# B&R Automation Studio project TrackingSample
Automation Studio 4.10.2.37; technology packages: mappCockpit 5.16.7002, mappMotion 5.16.7500, mappView 5.16.7001

## Configuration Cfg1

CPU 5PC900.TS17-00, AutomationRuntime B4.82, Build 6.3.0, Safety 1.10, Vc V4.33.0

### Task classes (Cpu.sw)
```
Cyclic#1 (cycle 1600 us, tolerance 0 us):
  DeltaCtrl <- Source.Motion.DeltaCtrl.prg
  ConveyorA <- Source.Motion.ConveyorA.prg
  ConveyorB <- Source.Motion.ConveyorB.prg
  ProductDet <- Source.Motion.ProductDetect.prg
  ProductPla <- Source.Motion.ProductPlacement.prg
  Program1 <- (binary)
  ServerP <- (binary)
  ServerR <- (binary)
  UN_Contro2 <- (binary)
DataObjects: McAcpSys, assl1
NcDataObjects: McDriveLog, mainCam, mainCam2, Cam
Binaries: TCData, udbdef, mcacpdrv, McMechSys, McAcpSim, McProfGen, arsvcreg, ArFlatPrv, ArCoal, McPathXT, mvLoader, mCoWebSc, Config_1, ashwd, sysconf, ashwac, asfw, arconfig, Role, iomap, User, Hierarchy, Rob1Ax, CodLim, Rob1AxGr4, CodMec4, Settings, Config, Config_7, Conveyor, CodMec, CodAxGr, Rob1AxGr, Config_5, Config_2, TCLang, Wr_Histor, Al_History, Al_Core, Wr_Core, GroupCore, Ev_Core, TraceConfi, Vis, TriggerCfg, ShuttleCfg, SectorCfg, AssemblyCf, asiol3, Vtrak, TC, User_1, asiol2, FifthAxCfg, PlowHeight, asnxdb3, viApp, Settings_1, viApp2, viApp1, viComp, asiol1, Config_3, asnxdb2, Cod_AxGr, Cod_Lim, Cod_Mec, Rob1_AxGr, Rob1_Ax, asiol4, OpcUaMap, asnxdb1, TriggCfg, Cams, Features, Webx_1, AssemblyCfg, Config_4, UNA, EM00, EM01, EMG, EMA, UN, EM00G, EM00A, EM01G, EM01A, PML
Libraries: DataObj, standard, runtime, astime, MpBase, AsArSdm, asstring, AsBrStr, MTTypes, brsystem, MTFilter, sys_lib, McBase, McAcpTrak, McAxis, McAcpPar, MpAxis, McAcpAx, CamProf, McPureVAx, MTBasics, AsIecCon, powerlnk, AsBrMath, BRIT_Data, MpRobotics, McAxGroup, McPathGen, McProgInt, AsIODiag, McTrkPath, MpPick, McPathSvc, CoTrace, AsZip, FileIO, asarprof, asarlog, AsMem, AsEPL, arssl, AsIO, aruser, ViBase, AsXml, AsTCP, SIKODrvLib, AcpInvLib, AsIOAcc, RVCarousel, AsSafety, MpServer, R_Lib_PM, AsHttp, MpRecipe, R_Lib, AsARCfg, R_Lib_Trak, R_PkML, MpPackML, MpAlarmX, ArUnitText, R_Siko, R_Carousel, areventlog
```

### Hardware
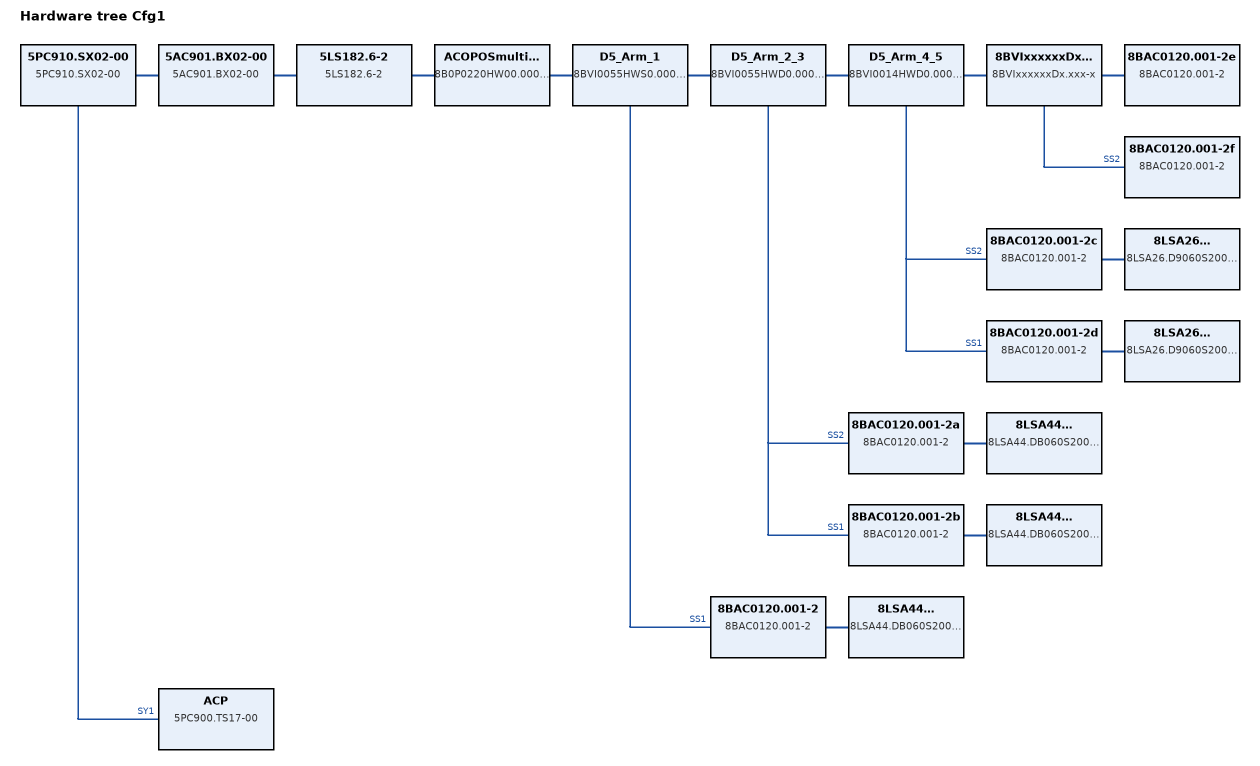
```
5AC901.BX02-00 : 5AC901.BX02-00 v1.0.1.0  [SY -> 5PC910.SX02-00.SY3]
5LS182.6-2 : 5LS182.6-2 v1.7.0.0  [SL -> 5AC901.BX02-00.SL1]
  Connector IF1:
    MtuSize = 1500
    DNAConfiguration = manual
    CycleTime = 1600
    EplNatSubnet = 192.168.102.0
    Channel1
    ChannelID1 = McAcpBroadcast
    ChannelType1 = OCTET[40]
    InternetAddress = 192.168.200.240
    SubnetMask = 255.255.255.0
5PC910.SX02-00 : 5PC910.SX02-00 v2.0.3.0
  Connector IF1:
    AssignedOperatingSystem = ARemb
  Connector IF3:
    AssignedOperatingSystem = ARemb
    ActivateDevice = 1
    Mode = Manual
    InternetAddress = 192.168.150.227
    SubnetMask = 255.255.255.0
  Connector IF4:
    AssignedOperatingSystem = ARemb
    ActivateDevice = 1
    Mode = Manual
    InternetAddress = 192.168.13.2
    SubnetMask = 255.255.255.0
  Connector IF5:
    AssignedOperatingSystem = ARemb
  Connector IF6:
    AssignedOperatingSystem = ARemb
  Connector IF7:
    AssignedOperatingSystem = ARemb
  Connector IF8:
    AssignedOperatingSystem = ARemb
  Connector IF9:
    AssignedOperatingSystem = ARemb
8BAC0120.001-2 : 8BAC0120.001-2 v2.2.0.0  [SS -> D5_Arm_1.SS1]
  PlugInType = Encoder
  McAcoposTypeID = AcoposMultiPlugInConfig
8BAC0120.001-2a : 8BAC0120.001-2 v2.2.0.0  [SS -> D5_Arm_2_3.SS2]
  PlugInType = Encoder
  McAcoposTypeID = AcoposMultiPlugInConfig
8BAC0120.001-2b : 8BAC0120.001-2 v2.2.0.0  [SS -> D5_Arm_2_3.SS1]
  PlugInType = Encoder
  McAcoposTypeID = AcoposMultiPlugInConfig
8BAC0120.001-2c : 8BAC0120.001-2 v2.2.0.0  [SS -> D5_Arm_4_5.SS2]
  PlugInType = Encoder
  McAcoposTypeID = AcoposMultiPlugInConfig
8BAC0120.001-2d : 8BAC0120.001-2 v2.2.0.0  [SS -> D5_Arm_4_5.SS1]
  PlugInType = Encoder
  McAcoposTypeID = AcoposMultiPlugInConfig
8BAC0120.001-2e : 8BAC0120.001-2 v2.2.0.0  [SS -> 8BVIxxxxxxDx.xxx-x2.SS1]
  PlugInType = Encoder
  McAcoposTypeID = AcoposMultiPlugInConfig
8BAC0120.001-2f : 8BAC0120.001-2 v2.2.0.0  [SS -> 8BVIxxxxxxDx.xxx-x2.SS2]
  PlugInType = Encoder
  McAcoposTypeID = AcoposMultiPlugInConfig
8BVIxxxxxxDx.xxx-x2 : 8BVIxxxxxxDx.xxx-x v2.3.0.0  [PLK1 -> D5_Arm_4_5.PLK2 (NodeNumber=7) [Cable Type=PowerlinkCable, Length=10, Version=1.0.0.3]]
  OrderNumber = 8BVI0014HWD0.000-1
  DriveConfiguration/Module:
    McAcoposTypeID = AcoposMultiDConfig
    ActivateACOPOSSimulationOnPLC = 0
    PowerSupply = DCBusVoltage
  DriveConfiguration/Module/PowerSupply:
    BusVoltage = 550
  DriveConfiguration/Channel[1]/RealAxis:
    AxisReference = gAxisConvB
  DriveConfiguration/Channel[1]/RealAxis/MechanicalElements/Gearbox:
    InputIsReadOnly = 0
    Input = 1
    OutputIsReadOnly = 0
    Output = 10
  DriveConfiguration/Channel[1]/RealAxis/MechanicalElements/RotaryToLinearTransformation:
    ReferenceDistanceIsReadOnly = 0
    ReferenceDistance = 3
  DriveConfiguration/Channel[1]/RealAxis/Controller:
    ModeIsReadOnly = 0
    Mode = PositionController
  DriveConfiguration/Channel[1]/RealAxis/Controller/Mode/Position:
    ProportionalGain = 460
    IntegrationTime = 0.0
    PredictionTime = 0.0004
    TotalDelayTime = 0.0004
  DriveConfiguration/Channel[1]/RealAxis/Controller/Mode/Speed:
    ProportionalGainIsReadOnly = 0
    ProportionalGain = 0.6
    IntegrationTimeIsReadOnly = 0
    IntegrationTime = 0.0
    FilterTimeIsReadOnly = 0
    FilterTime = 0.0
  DriveConfiguration/Channel[1]/RealAxis/Controller/Mode/LoopFilters:
    LoopFilter1 = NotUsed
    LoopFilter2 = NotUsed
    LoopFilter3 = NotUsed
  DriveConfiguration/Channel[1]/RealAxis/Homing:
    Mode = Direct
  DriveConfiguration/Channel[1]/RealAxis/Homing/Mode:
    Position = 0.0
    ReferencePulse = NotUsed
  DriveConfiguration/Channel[1]/RealAxis/Homing:
    RestorePositionVariable = 
  DriveConfiguration/Channel[1]/RealAxis/StopReaction:
    Quickstop = DecelerationLimit
    DriveError = DecelerationLimit
  DriveConfiguration/Channel[1]/RealAxis/MovementErrorLimits:
    PositionError = 1.0
    VelocityErrorMonitoring = Automatic1
  DriveConfiguration/Channel[1]/RealAxis:
    JerkFilter = NotUsed
  DriveConfiguration/Channel[1]/RealAxis/DigitalInputs/HomingSwitch:
    Source = NotUsed
    Level = High
  DriveConfiguration/Channel[1]/RealAxis/DigitalInputs/PositiveLimitSwitch:
    Source = NotUsed
    Level = High
  DriveConfiguration/Channel[1]/RealAxis/DigitalInputs/NegativeLimitSwitch:
    Source = NotUsed
    Level = High
  DriveConfiguration/Channel[1]/RealAxis/DigitalInputs/Trigger1:
    Source = X2Trigger1
    Level = High
  DriveConfiguration/Channel[1]/RealAxis/DigitalInputs/Trigger2:
    Source = X2Trigger2
    Level = High
  DriveConfiguration/Channel[1]/RealAxis/DigitalInputs/Quickstop:
    Input = Trigger2
  DriveConfiguration/Channel[1]/RealAxis/Simulation:
    SimulationModeOnPLC = SetValueGeneration
    SimulationModeOnACOPOS = NotUsed
  DriveConfiguration/Channel[1]:
    ExternalEncoderAxis = NotUsed
  DriveConfiguration/Channel[2]/RealAxis:
    AxisReference = gAxisConvA
  DriveConfiguration/Channel[2]/RealAxis/MechanicalElements/Gearbox:
    InputIsReadOnly = 0
    Input = 1
    OutputIsReadOnly = 0
    Output = 10
  DriveConfiguration/Channel[2]/RealAxis/MechanicalElements/RotaryToLinearTransformation:
    ReferenceDistanceIsReadOnly = 0
    ReferenceDistance = 3
  DriveConfiguration/Channel[2]/RealAxis/Controller:
    ModeIsReadOnly = 0
    Mode = PositionController
  DriveConfiguration/Channel[2]/RealAxis/Controller/Mode/Position:
    ProportionalGain = 435
    IntegrationTime = 0.0
    PredictionTime = 0.0004
    TotalDelayTime = 0.0004
  DriveConfiguration/Channel[2]/RealAxis/Controller/Mode/Speed:
    ProportionalGainIsReadOnly = 0
    ProportionalGain = 0.55
    IntegrationTimeIsReadOnly = 0
    IntegrationTime = 0.0
    FilterTimeIsReadOnly = 0
    FilterTime = 0.0
  DriveConfiguration/Channel[2]/RealAxis/Controller/Mode/LoopFilters:
    LoopFilter1 = NotUsed
    LoopFilter2 = NotUsed
    LoopFilter3 = NotUsed
  DriveConfiguration/Channel[2]/RealAxis/Homing:
    Mode = Direct
  DriveConfiguration/Channel[2]/RealAxis/Homing/Mode:
    Position = 0.0
    ReferencePulse = NotUsed
  DriveConfiguration/Channel[2]/RealAxis/Homing:
    RestorePositionVariable = 
  DriveConfiguration/Channel[2]/RealAxis/StopReaction:
    Quickstop = DecelerationLimit
    DriveError = DecelerationLimit
  DriveConfiguration/Channel[2]/RealAxis/MovementErrorLimits:
    PositionError = 1.0
    VelocityErrorMonitoring = Automatic1
  DriveConfiguration/Channel[2]/RealAxis:
    JerkFilter = NotUsed
  DriveConfiguration/Channel[2]/RealAxis/DigitalInputs/HomingSwitch:
    Source = NotUsed
    Level = High
  DriveConfiguration/Channel[2]/RealAxis/DigitalInputs/PositiveLimitSwitch:
    Source = NotUsed
    Level = High
  DriveConfiguration/Channel[2]/RealAxis/DigitalInputs/NegativeLimitSwitch:
    Source = NotUsed
    Level = High
  DriveConfiguration/Channel[2]/RealAxis/DigitalInputs/Trigger1:
    Source = X2Trigger1
    Level = High
  DriveConfiguration/Channel[2]/RealAxis/DigitalInputs/Trigger2:
    Source = X2Trigger2
    Level = High
  DriveConfiguration/Channel[2]/RealAxis/DigitalInputs/Quickstop:
    Input = Trigger2
  DriveConfiguration/Channel[2]/RealAxis/Simulation:
    SimulationModeOnPLC = SetValueGeneration
    SimulationModeOnACOPOS = NotUsed
  DriveConfiguration/Channel[2]:
    ExternalEncoderAxis = NotUsed
8LSA26.D9060S200-3 : 8LSA26.D9060S200-3 v1.0.7.40  [EC -> 8BAC0120.001-2d.EC; MT -> D5_Arm_4_5.MT1]
8LSA26.D9060S200-3a : 8LSA26.D9060S200-3 v1.0.7.40  [EC -> 8BAC0120.001-2c.EC; MT -> D5_Arm_4_5.MT2]
8LSA44.DB060S200-3 : 8LSA44.DB060S200-3 v1.0.9.37  [EC -> 8BAC0120.001-2.EC; MT -> D5_Arm_1.MT1]
8LSA44.DB060S200-3a : 8LSA44.DB060S200-3 v1.0.9.37  [EC -> 8BAC0120.001-2a.EC; MT -> D5_Arm_2_3.MT2]
8LSA44.DB060S200-3b : 8LSA44.DB060S200-3 v1.0.9.37  [EC -> 8BAC0120.001-2b.EC; MT -> D5_Arm_2_3.MT1]
ACOPOSmulti_Rack_PS : 8B0P0220HW00.000-1 v2.3.0.0  [PLK1 -> 5LS182.6-2.IF1 (NodeNumber=100) [Cable Type=PowerlinkCable, Length=10, Version=1.0.0.3]; PLK2 -> D5_Arm_1.PLK1 (NodeNumber=100) [Cable Type=PowerlinkCable, Length=10, Version=1.0.0.3]]
  DriveConfiguration/Module:
    McAcoposTypeID = AcoposMultiPSMpConfig
    ActivateACOPOSSimulationOnPLC = 0
  DriveConfiguration/Channel[1]/PowerSection:
    AxisReference = gRobPS
  DriveConfiguration/Channel[1]/ChannelFeatures:
    FeatureRef[1] = Feature_AcpParTable
ACP : 5PC900.TS17-00 v2.1.0.0  [SY -> 5PC910.SX02-00.SY1]
  ConfigurationID = Betel
  UserPartitionSize = 10
  Simulation = 1
  RemMemDevice = PCI.1.LS182.SRAM
  RemMemSize = 10000
  PermanentPvSize = 9000
  RemanentGlobalPvSize = 100
  VolatileGlobalPvSize = 4000000
  ClearNVMemoryAfterCFChange = 1
  TimerDeviceType = EPLX2X
  TimerDevice = 5LS182.6-2.IF1
  IdleTaskClass = 4
  TaskClassIdleTime = 3200
  Cyclic1Duration = 1600
  Cyclic1Tolerance = 0
  Cyclic1Stack = 1000000
  Cyclic1Output = 1
  Cyclic2Duration = 19200
  Cyclic2Tolerance = 19200
  Cyclic3Duration = 48000
  Cyclic3Tolerance = 48000
  Cyclic4Duration = 99200
  Cyclic4Tolerance = 99200
  Cyclic6Duration = 499200
  Cyclic6Tolerance = 499200
  Cyclic8Duration = 16000
  FileDevice1
  FileDeviceName1 = CNC_Programs
  FileDevicePath1 = C:\projects\MCR\TrackingSample\Logical\Source\Motion\RobotProgram
  TimeZone = 140
  ActivateDaylightSavingTime = 1
  FtpUser1
  FtpUsername1 = ronchi
  FtpUserPassword1 = Qr4mnGyRDGFj5/UnqR7ZzE2TygV13U3viQDWrGQj2Tc=
  FtpUserSalt1 = 2ZufkTNm
  FTPAccessRight1 = 0
  ActivateOpcUa = 1
  OpcUa_AuthenticationSecurityPolicy_EnableNone = 1
  OpcUa_AuthenticationSecurityPolicy_EnableBasic128Rsa15 = 1
  OpcUa_Security_AdminRole = Everyone
  OpcUa_Limits_MonitoredItemsPerSubscription = 5000
  OpcUaMaxSubsEventQueueSize = 5000
  OpcUaInformationModels_PV_Version = 1
D5_Arm_1 : 8BVI0055HWS0.000-1 v2.2.0.0  [PLK1 -> ACOPOSmulti_Rack_PS.PLK2 [Cable Type=PowerlinkCable, Length=10, Version=1.0.0.3]; PLK2 -> D5_Arm_2_3.PLK1 [Cable Type=PowerlinkCable, Length=10, Version=1.0.0.3]]
  DriveConfiguration/Module:
    McAcoposTypeID = AcoposMultiDConfig
    ActivateACOPOSSimulationOnPLC = 0
  DriveConfiguration/Module/PowerSupply:
    PowerSupplyModuleReference = gRobPS
  DriveConfiguration/Channel[1]/RealAxis:
    AxisReference = gR1_AxisQ1
  DriveConfiguration/Channel[1]/RealAxis/MechanicalElements/Gearbox:
    InputIsReadOnly = 0
    Input = 31
    OutputIsReadOnly = 0
    Output = 1
  DriveConfiguration/Channel[1]/RealAxis/MechanicalElements/RotaryToLinearTransformation:
    ReferenceDistanceIsReadOnly = 0
    ReferenceDistance = 1
  DriveConfiguration/Channel[1]/RealAxis/Controller:
    ModeIsReadOnly = 0
    Mode = PositionController
  DriveConfiguration/Channel[1]/RealAxis/Controller/Mode/Position:
    ProportionalGain = 150
    IntegrationTime = 0.0
    PredictionTime = 0.0004
    TotalDelayTime = 0.0004
  DriveConfiguration/Channel[1]/RealAxis/Controller/Mode/Speed:
    ProportionalGainIsReadOnly = 0
    ProportionalGain = 5
    IntegrationTimeIsReadOnly = 0
    IntegrationTime = 0.0
    FilterTimeIsReadOnly = 0
    FilterTime = 0.0
  DriveConfiguration/Channel[1]/RealAxis/Controller/Mode/LoopFilters:
    LoopFilter1 = NotUsed
    LoopFilter2 = NotUsed
    LoopFilter3 = NotUsed
  DriveConfiguration/Channel[1]/RealAxis/Homing:
    Mode = RestorePosition
    RestorePositionVariable = ::HomePos_R1[0]
  DriveConfiguration/Channel[1]/RealAxis/StopReaction:
    Quickstop = DecelerationLimit
    DriveError = DecelerationLimit
  DriveConfiguration/Channel[1]/RealAxis/MovementErrorLimits:
    PositionError = 1.0
    VelocityErrorMonitoring = Automatic1
  DriveConfiguration/Channel[1]/RealAxis:
    JerkFilter = Used
  DriveConfiguration/Channel[1]/RealAxis/JerkFilter:
    JerkTime = 0.02
  DriveConfiguration/Channel[1]/RealAxis/DigitalInputs/HomingSwitch:
    Source = NotUsed
    Level = High
  DriveConfiguration/Channel[1]/RealAxis/DigitalInputs/PositiveLimitSwitch:
    Source = NotUsed
    Level = High
  DriveConfiguration/Channel[1]/RealAxis/DigitalInputs/NegativeLimitSwitch:
    Source = NotUsed
    Level = High
  DriveConfiguration/Channel[1]/RealAxis/DigitalInputs/Trigger1:
    Level = High
  DriveConfiguration/Channel[1]/RealAxis/DigitalInputs/Trigger2:
    Level = High
  DriveConfiguration/Channel[1]/RealAxis/DigitalInputs/Quickstop:
    Input = Trigger2
  DriveConfiguration/Channel[1]/RealAxis/Simulation:
    SimulationModeOnPLC = SetValueGeneration
    SimulationModeOnACOPOS = NotUsed
  DriveConfiguration/Channel[2]/RealAxis:
    AxisReference = 
  DriveConfiguration/Channel[2]/RealAxis/MechanicalElements/Gearbox:
    InputIsReadOnly = 0
    Input = 1
    OutputIsReadOnly = 0
    Output = 1
  DriveConfiguration/Channel[2]/RealAxis/MechanicalElements/RotaryToLinearTransformation:
    ReferenceDistanceIsReadOnly = 0
    ReferenceDistance = 1
  DriveConfiguration/Channel[2]/RealAxis/Controller:
    ModeIsReadOnly = 0
    Mode = PositionController
  DriveConfiguration/Channel[2]/RealAxis/Controller/Mode/Position:
    ProportionalGain = 50.0
    IntegrationTime = 0.0
    PredictionTime = 0.0004
    TotalDelayTime = 0.0004
  DriveConfiguration/Channel[2]/RealAxis/Controller/Mode/Speed:
    ProportionalGainIsReadOnly = 0
    ProportionalGain = 2.0
    IntegrationTimeIsReadOnly = 0
    IntegrationTime = 0.0
    FilterTimeIsReadOnly = 0
    FilterTime = 0.0
  DriveConfiguration/Channel[2]/RealAxis/Controller/Mode/LoopFilters:
    LoopFilter1 = NotUsed
    LoopFilter2 = NotUsed
    LoopFilter3 = NotUsed
  DriveConfiguration/Channel[2]/RealAxis/Homing:
    Mode = Direct
  DriveConfiguration/Channel[2]/RealAxis/Homing/Mode:
    Position = 0.0
    ReferencePulse = NotUsed
  DriveConfiguration/Channel[2]/RealAxis/Homing:
    RestorePositionVariable = 
  DriveConfiguration/Channel[2]/RealAxis/StopReaction:
    Quickstop = DecelerationLimit
    DriveError = DecelerationLimit
  DriveConfiguration/Channel[2]/RealAxis/MovementErrorLimits:
    PositionError = 1.0
    VelocityErrorMonitoring = Automatic1
  DriveConfiguration/Channel[2]/RealAxis:
    JerkFilter = NotUsed
  DriveConfiguration/Channel[2]/RealAxis/DigitalInputs/HomingSwitch:
    Source = NotUsed
    Level = High
  DriveConfiguration/Channel[2]/RealAxis/DigitalInputs/PositiveLimitSwitch:
    Source = NotUsed
    Level = High
  DriveConfiguration/Channel[2]/RealAxis/DigitalInputs/NegativeLimitSwitch:
    Source = NotUsed
    Level = High
  DriveConfiguration/Channel[2]/RealAxis/DigitalInputs/Trigger1:
    Level = High
  DriveConfiguration/Channel[2]/RealAxis/DigitalInputs/Trigger2:
    Level = High
  DriveConfiguration/Channel[2]/RealAxis/DigitalInputs/Quickstop:
    Input = Trigger2
  DriveConfiguration/Channel[2]/RealAxis/Simulation:
    SimulationModeOnPLC = SetValueGeneration
    SimulationModeOnACOPOS = NotUsed
D5_Arm_2_3 : 8BVI0055HWD0.000-1 v2.2.0.0  [PLK1 -> D5_Arm_1.PLK2 [Cable Type=PowerlinkCable, Length=10, Version=1.0.0.3]; PLK2 -> D5_Arm_4_5.PLK1 [Cable Type=PowerlinkCable, Length=10, Version=1.0.0.3]; MT2 -> 8LSA44.DB060S200-3a.MT]
  DriveConfiguration/Module:
    McAcoposTypeID = AcoposMultiDConfig
    ActivateACOPOSSimulationOnPLC = 0
  DriveConfiguration/Module/PowerSupply:
    PowerSupplyModuleReference = gRobPS
  DriveConfiguration/Channel[1]/RealAxis:
    AxisReference = gR1_AxisQ3
  DriveConfiguration/Channel[1]/RealAxis/MechanicalElements/Gearbox:
    InputIsReadOnly = 0
    Input = 31
    OutputIsReadOnly = 0
    Output = 1
  DriveConfiguration/Channel[1]/RealAxis/MechanicalElements/RotaryToLinearTransformation:
    ReferenceDistanceIsReadOnly = 0
    ReferenceDistance = 1
  DriveConfiguration/Channel[1]/RealAxis/Controller:
    ModeIsReadOnly = 0
    Mode = PositionController
  DriveConfiguration/Channel[1]/RealAxis/Controller/Mode/Position:
    ProportionalGain = 150
    IntegrationTime = 0.0
    PredictionTime = 0.0004
    TotalDelayTime = 0.0004
  DriveConfiguration/Channel[1]/RealAxis/Controller/Mode/Speed:
    ProportionalGainIsReadOnly = 0
    ProportionalGain = 5
    IntegrationTimeIsReadOnly = 0
    IntegrationTime = 0.0
    FilterTimeIsReadOnly = 0
    FilterTime = 0.0
  DriveConfiguration/Channel[1]/RealAxis/Controller/Mode/LoopFilters:
    LoopFilter1 = NotUsed
    LoopFilter2 = NotUsed
    LoopFilter3 = NotUsed
  DriveConfiguration/Channel[1]/RealAxis/Homing:
    Mode = RestorePosition
    RestorePositionVariable = ::HomePos_R1[2]
  DriveConfiguration/Channel[1]/RealAxis/StopReaction:
    Quickstop = DecelerationLimit
    DriveError = DecelerationLimit
  DriveConfiguration/Channel[1]/RealAxis/MovementErrorLimits:
    PositionError = 1.0
    VelocityErrorMonitoring = Automatic1
  DriveConfiguration/Channel[1]/RealAxis:
    JerkFilter = Used
  DriveConfiguration/Channel[1]/RealAxis/JerkFilter:
    JerkTime = 0.02
  DriveConfiguration/Channel[1]/RealAxis/DigitalInputs/HomingSwitch:
    Source = NotUsed
    Level = High
  DriveConfiguration/Channel[1]/RealAxis/DigitalInputs/PositiveLimitSwitch:
    Source = NotUsed
    Level = High
  DriveConfiguration/Channel[1]/RealAxis/DigitalInputs/NegativeLimitSwitch:
    Source = NotUsed
    Level = High
  DriveConfiguration/Channel[1]/RealAxis/DigitalInputs/Trigger1:
    Level = High
  DriveConfiguration/Channel[1]/RealAxis/DigitalInputs/Trigger2:
    Level = High
  DriveConfiguration/Channel[1]/RealAxis/DigitalInputs/Quickstop:
    Input = Trigger2
  DriveConfiguration/Channel[1]/RealAxis/Simulation:
    SimulationModeOnPLC = SetValueGeneration
    SimulationModeOnACOPOS = NotUsed
  DriveConfiguration/Channel[2]/RealAxis:
    AxisReference = gR1_AxisQ2
  DriveConfiguration/Channel[2]/RealAxis/MechanicalElements/Gearbox:
    InputIsReadOnly = 0
    Input = 31
    OutputIsReadOnly = 0
    Output = 1
  DriveConfiguration/Channel[2]/RealAxis/MechanicalElements/RotaryToLinearTransformation:
    ReferenceDistanceIsReadOnly = 0
    ReferenceDistance = 1
  DriveConfiguration/Channel[2]/RealAxis/Controller:
    ModeIsReadOnly = 0
    Mode = PositionController
  DriveConfiguration/Channel[2]/RealAxis/Controller/Mode/Position:
    ProportionalGain = 150
    IntegrationTime = 0.0
    PredictionTime = 0.0004
    TotalDelayTime = 0.0004
  DriveConfiguration/Channel[2]/RealAxis/Controller/Mode/Speed:
    ProportionalGainIsReadOnly = 0
    ProportionalGain = 5
    IntegrationTimeIsReadOnly = 0
    IntegrationTime = 0.0
    FilterTimeIsReadOnly = 0
    FilterTime = 0.0
  DriveConfiguration/Channel[2]/RealAxis/Controller/Mode/LoopFilters:
    LoopFilter1 = NotUsed
    LoopFilter2 = NotUsed
    LoopFilter3 = NotUsed
  DriveConfiguration/Channel[2]/RealAxis/Homing:
    Mode = RestorePosition
    RestorePositionVariable = ::HomePos_R1[1]
  DriveConfiguration/Channel[2]/RealAxis/StopReaction:
    Quickstop = DecelerationLimit
    DriveError = DecelerationLimit
  DriveConfiguration/Channel[2]/RealAxis/MovementErrorLimits:
    PositionError = 1.0
    VelocityErrorMonitoring = Automatic1
  DriveConfiguration/Channel[2]/RealAxis:
    JerkFilter = Used
  DriveConfiguration/Channel[2]/RealAxis/JerkFilter:
    JerkTime = 0.02
  DriveConfiguration/Channel[2]/RealAxis/DigitalInputs/HomingSwitch:
    Source = NotUsed
    Level = High
  DriveConfiguration/Channel[2]/RealAxis/DigitalInputs/PositiveLimitSwitch:
    Source = NotUsed
    Level = High
  DriveConfiguration/Channel[2]/RealAxis/DigitalInputs/NegativeLimitSwitch:
    Source = NotUsed
    Level = High
  DriveConfiguration/Channel[2]/RealAxis/DigitalInputs/Trigger1:
    Level = High
  DriveConfiguration/Channel[2]/RealAxis/DigitalInputs/Trigger2:
    Level = High
  DriveConfiguration/Channel[2]/RealAxis/DigitalInputs/Quickstop:
    Input = Trigger2
  DriveConfiguration/Channel[2]/RealAxis/Simulation:
    SimulationModeOnPLC = SetValueGeneration
    SimulationModeOnACOPOS = NotUsed
D5_Arm_4_5 : 8BVI0014HWD0.000-1 v2.2.0.0  [PLK1 -> D5_Arm_2_3.PLK2 [Cable Type=PowerlinkCable, Length=10, Version=1.0.0.3]; PLK2 -> 8BVIxxxxxxDx.xxx-x2.PLK1 [Cable Type=PowerlinkCable, Length=10, Version=1.0.0.3]; MT2 -> 8LSA26.D9060S200-3a.MT]
  DriveConfiguration/Module:
    McAcoposTypeID = AcoposMultiDConfig
    ActivateACOPOSSimulationOnPLC = 0
  DriveConfiguration/Module/PowerSupply:
    PowerSupplyModuleReference = gRobPS
  DriveConfiguration/Channel[1]/RealAxis:
    AxisReference = gR1_AxisQC
  DriveConfiguration/Channel[1]/RealAxis/MechanicalElements/Gearbox:
    InputIsReadOnly = 0
    Input = 20
    OutputIsReadOnly = 0
    Output = 1
  DriveConfiguration/Channel[1]/RealAxis/MechanicalElements/RotaryToLinearTransformation:
    ReferenceDistanceIsReadOnly = 0
    ReferenceDistance = 1
  DriveConfiguration/Channel[1]/RealAxis/Controller:
    ModeIsReadOnly = 0
    Mode = PositionController
  DriveConfiguration/Channel[1]/RealAxis/Controller/Mode/Position:
    ProportionalGain = 150
    IntegrationTime = 0.0
    PredictionTime = 0.0004
    TotalDelayTime = 0.0004
  DriveConfiguration/Channel[1]/RealAxis/Controller/Mode/Speed:
    ProportionalGainIsReadOnly = 0
    ProportionalGain = 0.6
    IntegrationTimeIsReadOnly = 0
    IntegrationTime = 0.0
    FilterTimeIsReadOnly = 0
    FilterTime = 0.0
  DriveConfiguration/Channel[1]/RealAxis/Controller/Mode/LoopFilters:
    LoopFilter1 = NotUsed
    LoopFilter2 = NotUsed
    LoopFilter3 = NotUsed
  DriveConfiguration/Channel[1]/RealAxis/Homing:
    Mode = RestorePosition
    RestorePositionVariable = ::HomePos_R1[3]
  DriveConfiguration/Channel[1]/RealAxis/StopReaction:
    Quickstop = DecelerationLimit
    DriveError = DecelerationLimit
  DriveConfiguration/Channel[1]/RealAxis/MovementErrorLimits:
    PositionError = 1.0
    VelocityErrorMonitoring = Automatic1
  DriveConfiguration/Channel[1]/RealAxis:
    JerkFilter = Used
  DriveConfiguration/Channel[1]/RealAxis/JerkFilter:
    JerkTime = 0.01
  DriveConfiguration/Channel[1]/RealAxis/DigitalInputs/HomingSwitch:
    Source = NotUsed
    Level = High
  DriveConfiguration/Channel[1]/RealAxis/DigitalInputs/PositiveLimitSwitch:
    Source = NotUsed
    Level = High
  DriveConfiguration/Channel[1]/RealAxis/DigitalInputs/NegativeLimitSwitch:
    Source = NotUsed
    Level = High
  DriveConfiguration/Channel[1]/RealAxis/DigitalInputs/Trigger1:
    Level = High
  DriveConfiguration/Channel[1]/RealAxis/DigitalInputs/Trigger2:
    Level = High
  DriveConfiguration/Channel[1]/RealAxis/DigitalInputs/Quickstop:
    Input = Trigger2
  DriveConfiguration/Channel[1]/RealAxis/Simulation:
    SimulationModeOnPLC = SetValueGeneration
    SimulationModeOnACOPOS = NotUsed
  DriveConfiguration/Channel[2]/RealAxis:
    AxisReference = gR1_AxisQA
  DriveConfiguration/Channel[2]/RealAxis/MechanicalElements/Gearbox:
    InputIsReadOnly = 0
    Input = 20
    OutputIsReadOnly = 0
    Output = 1
  DriveConfiguration/Channel[2]/RealAxis/MechanicalElements/RotaryToLinearTransformation:
    ReferenceDistanceIsReadOnly = 0
    ReferenceDistance = 1
  DriveConfiguration/Channel[2]/RealAxis/Controller:
    ModeIsReadOnly = 0
    Mode = PositionController
  DriveConfiguration/Channel[2]/RealAxis/Controller/Mode/Position:
    ProportionalGain = 150
    IntegrationTime = 0.0
    PredictionTime = 0.0004
    TotalDelayTime = 0.0004
  DriveConfiguration/Channel[2]/RealAxis/Controller/Mode/Speed:
    ProportionalGainIsReadOnly = 0
    ProportionalGain = 0.6
    IntegrationTimeIsReadOnly = 0
    IntegrationTime = 0.0
    FilterTimeIsReadOnly = 0
    FilterTime = 0.0
  DriveConfiguration/Channel[2]/RealAxis/Controller/Mode/LoopFilters:
    LoopFilter1 = NotUsed
    LoopFilter2 = NotUsed
    LoopFilter3 = NotUsed
  DriveConfiguration/Channel[2]/RealAxis/Homing:
    Mode = RestorePosition
    RestorePositionVariable = ::HomePos_R1[4]
  DriveConfiguration/Channel[2]/RealAxis/StopReaction:
    Quickstop = DecelerationLimit
    DriveError = DecelerationLimit
  DriveConfiguration/Channel[2]/RealAxis/MovementErrorLimits:
    PositionError = 1.0
    VelocityErrorMonitoring = Automatic1
  DriveConfiguration/Channel[2]/RealAxis:
    JerkFilter = Used
  DriveConfiguration/Channel[2]/RealAxis/JerkFilter:
    JerkTime = 0.01
  DriveConfiguration/Channel[2]/RealAxis/DigitalInputs/HomingSwitch:
    Source = NotUsed
    Level = High
  DriveConfiguration/Channel[2]/RealAxis/DigitalInputs/PositiveLimitSwitch:
    Source = NotUsed
    Level = High
  DriveConfiguration/Channel[2]/RealAxis/DigitalInputs/NegativeLimitSwitch:
    Source = NotUsed
    Level = High
  DriveConfiguration/Channel[2]/RealAxis/DigitalInputs/Trigger1:
    Level = High
  DriveConfiguration/Channel[2]/RealAxis/DigitalInputs/Trigger2:
    Level = High
  DriveConfiguration/Channel[2]/RealAxis/DigitalInputs/Quickstop:
    Input = Trigger2
  DriveConfiguration/Channel[2]/RealAxis/Simulation:
    SimulationModeOnPLC = SetValueGeneration
    SimulationModeOnACOPOS = NotUsed
```

### Config.mappmotioncfg - ACP/mappMotion/Config.mappmotioncfg
```
Element MappMotionConfiguration (Type=mappmotioncfg)
  Processing:
    ProcessingTaskClass = 1
  Logger:
    SelectiveLogging = Used
      AdministrativeCommands = Suppressed
      MovementCommands = Visible
      InformationalCommands = Suppressed
      SuppressSubcomponents = Inactive
```

### Config_5.axis - ACP/mappMotion/Config_5.axis
```
Element gAxisConvA (Type=axis)
  BaseTypeIsReadOnly = 0
  BaseType = LinearPeriodic
    MeasurementUnit = 5066068
    MeasurementResolutionIsReadOnly = 0
    MeasurementResolution = 0.001
    CountDirectionIsReadOnly = 0
    CountDirection = Standard
    PeriodSettings:
      Period = 1200
  MovementLimitsIsReadOnly = 0
  MovementLimits = Internal
    Position:
      LowerLimitMin = -1.79769313486231E308
      UpperLimitMax = 1.79769313486231E308
      LowerLimit = -1000.0
      UpperLimit = 1000.0
    VelocityIsReadOnly = 0
    Velocity:
      VelocityMax = 3.4E38
      Velocity = 2000
    AccelerationIsReadOnly = 0
    Acceleration:
      AccelerationMax = 3.4E38
      Acceleration = 5000
    DecelerationIsReadOnly = 0
    Deceleration:
      DecelerationMax = 3.4E38
      Deceleration = 5000
  Alarms = None
```

### Conveyor.axis - ACP/mappMotion/Conveyor.axis
```
Element gAxisConvB (Type=axis)
  BaseTypeIsReadOnly = 0
  BaseType = LinearPeriodic
    MeasurementUnit = 5066068
    MeasurementResolutionIsReadOnly = 0
    MeasurementResolution = 0.001
    CountDirectionIsReadOnly = 0
    CountDirection = Standard
    PeriodSettings:
      Period = 1200
  MovementLimitsIsReadOnly = 0
  MovementLimits = Internal
    Position:
      LowerLimitMin = -1.79769313486231E308
      UpperLimitMax = 1.79769313486231E308
      LowerLimit = -1000.0
      UpperLimit = 1000.0
    VelocityIsReadOnly = 0
    Velocity:
      VelocityMax = 3.4E38
      Velocity = 2000
    AccelerationIsReadOnly = 0
    Acceleration:
      AccelerationMax = 3.4E38
      Acceleration = 5000
    DecelerationIsReadOnly = 0
    Deceleration:
      DecelerationMax = 3.4E38
      Deceleration = 5000
  Alarms = None
Element gAxisConvA (Type=axis)
  BaseTypeIsReadOnly = 0
  BaseType = LinearPeriodic
    MeasurementUnit = 5066068
    MeasurementResolutionIsReadOnly = 0
    MeasurementResolution = 0.001
    CountDirectionIsReadOnly = 0
    CountDirection = Standard
    PeriodSettings:
      Period = 1200
  MovementLimitsIsReadOnly = 0
  MovementLimits = Internal
    Position:
      LowerLimitMin = -1.79769313486231E308
      UpperLimitMax = 1.79769313486231E308
      LowerLimit = -1000.0
      UpperLimit = 1000.0
    VelocityIsReadOnly = 0
    Velocity:
      VelocityMax = 3.4E38
      Velocity = 2000
    AccelerationIsReadOnly = 0
    Acceleration:
      AccelerationMax = 3.4E38
      Acceleration = 5000
    DecelerationIsReadOnly = 0
    Deceleration:
      DecelerationMax = 3.4E38
      Deceleration = 5000
  Alarms = None
```

### CodLim.limitset - ACP/mappMotion/Rob/Codian_4ax/CodLim.limitset
```
Element LimitArm (Type=limitset)
  Type = RotaryLimit
    Position = Used
      LowerLimitMin = -1.79769313486231E308
      UpperLimitMax = 1.79769313486231E308
      LowerLimit = -38.0
      UpperLimit = 88.0
    Velocity = Basic
      VelocityMax = 3.4E38
      Velocity = 5000
    Acceleration = Basic
      AccelerationMax = 3.4E38
      Acceleration = 50000.0
    Deceleration = Basic
      DecelerationMax = 3.4E38
      Deceleration = 50000.0
    JerkIsReadOnly = 0
    TorqueIsReadOnly = 0
Element LimitRotation (Type=limitset)
  Type = RotaryLimit
    Velocity = Basic
      VelocityMax = 3.4E38
      Velocity = 3600
    Acceleration = Basic
      AccelerationMax = 3.4E38
      Acceleration = 36000
    Deceleration = Basic
      DecelerationMax = 3.4E38
      Deceleration = 36000
    JerkIsReadOnly = 0
    TorqueIsReadOnly = 0
Element LimitTilt (Type=limitset)
  Type = RotaryLimit
    Velocity = Basic
      VelocityMax = 3.4E38
      Velocity = 3600
    Acceleration = Basic
      AccelerationMax = 3.4E38
      Acceleration = 36000
    Deceleration = Basic
      DecelerationMax = 3.4E38
      Deceleration = 36000
    JerkIsReadOnly = 0
    TorqueIsReadOnly = 0
```

### CodMec4.mechanicalsystem - ACP/mappMotion/Rob/Codian_4ax/CodMec4.mechanicalsystem
```
Element MechSys_4ax (Type=mechanicalsystem)
  Type = Delta
    Subtype = 4AxesDeltaA
      Description = Standard
        Dimensions:
          BasePlatform:
            CenterIsReadOnly = 0
            Center:
              X = 0.0
              Y = 0.0
              Z = 0.0
            ArmLinkPointIsReadOnly = 0
            Arm1LinkPoint:
              Angle = 0.0
              Radius = 200
              Z = -90
            Arm2LinkPoint:
              Angle = -120.0
              Radius = 200
              Z = -90
            Arm3LinkPoint:
              Angle = -240.0
              Radius = 200
              Z = -90
          Arms:
            ArmIsReadOnly = 0
            Arm1:
              UpperArmLength = 320
              LowerArmLength = 850
            Arm2:
              UpperArmLength = 320
              LowerArmLength = 850
            Arm3:
              UpperArmLength = 320
              LowerArmLength = 850
          EndEffectorPlatform:
            ArmLinkPointIsReadOnly = 0
            Arm1LinkPoint:
              Radius = 50
              Z = 0.0
            Arm2LinkPoint:
              Radius = 50
              Z = 0.0
            Arm3LinkPoint:
              Radius = 50
              Z = 0.0
            TranslationToFlange:
              X = 0.0
              Y = 0.0
              Z = -44.5
        Offsets:
          JointAxisIsReadOnly = 0
          JointAxis[1] = 0.0
          JointAxis[2] = 0.0
          JointAxis[3] = 0.0
          JointAxis[4] = 0.0
        CountDirections:
          JointAxisIsReadOnly = 0
          JointAxis[1] = Standard
          JointAxis[2] = Standard
          JointAxis[3] = Standard
          JointAxis[4] = Standard
      CoordinatesNames = Default
        XCoordinateName = X
        YCoordinateName = Y
        ZCoordinateName = Z
        CCoordinateName = C
      WireFrameModel = Standard
        UpperArm1 = ConnectionLine
          Distance = 0.0
        LowerArm1 = ConnectionLine
          Distance = 0.0
        UpperArm2 = ConnectionLine
          Distance = 0.0
        LowerArm2 = ConnectionLine
          Distance = 0.0
        UpperArm3 = ConnectionLine
          Distance = 0.0
        LowerArm3 = ConnectionLine
          Distance = 0.0
        EndEffectorPlatformToFlange = ConnectionLine
          Distance = 0.0
        FlangeToTcp = ConnectionLine
          Distance = 0.0
      DynamicModel = DynParTable
        TableRef
      InternalDynamicModel = NotUsed
      DynamicLimits = DynParTables
        GearboxLimitsTableRef
        CrossSectionLimitsTableRef
      InternalDynamicLimits = NotUsed
      JointAxesPositionLimits:
        JointAxis[1] = UseAxisLimits
        JointAxis[2] = UseAxisLimits
        JointAxis[3] = UseAxisLimits
        JointAxis[4] = UseAxisLimits
      WorkingRange = NotUsed
```

### Config_7.axesgroupfeature - ACP/mappMotion/Rob/Config_7.axesgroupfeature
```
Element Feature_FrameHierarchy (Type=axesgroupfeature)
  Type = FrameHierarchy
    ModalDataBehaviour = UseAxesGroupSettings
    FrameHierarchy = Custom
      FramePropertyMapping:
        BCS = RobotBase
        PCS = MachineFrame
        SCS1
        SCS2
        SCS3
        SCS4
        SCS5
      MCS:
        Frame[1]:
          Name = RobotBase
          Type = StandardFrame
            Translation:
              X = 0.0
              Y = 0.0
              Z = 0.0
            Orientation:
              Angle1 = 0.0
              Angle2 = 0.0
              Angle3 = 180
Element Feature_Jogging (Type=axesgroupfeature)
  Type = Jogging
Element Feature_Programs (Type=axesgroupfeature)
  Type = Program
    ModalDataBehaviour = UseAxesGroupSettings
    InitialSettings:
      InterpolationTypes = LinearRapid
      PositionCoordinates = Absolute
      CircleCoordinates = Relative
      JACS_ACSProgramming = JACS
      ContourConnection = Inactive
      ProgrammingUnits = UseAxesGroupSettings
      Feedrates:
        FeedPath = Standard
        FeedCharacteristic = StandardCharacteristic
        FeedType = Feedrate
        FeedReduction = Inactive
        FeedrateValue = 0.0
        InverseFeedrateValue = 0.0
        FeedratePerRevValue = 0.0
    DefaultLanguage = ST
    Location = User
      UserLocation[1]:
        FileDevice = CNC_Programs
    ProgramElements:
      PVs:
        PV[1]:
          PvName = ::gDeltaCtrl.Status.ProductPicked
          Advanced:
            Alias = ProductPicked
            Synchronization = Path
            Reference = No
        PV[2]:
          PvName = ::gDeltaCtrl.Status.ProductPlaced
          Advanced:
            Alias = ProductPlaced
            Synchronization = Path
            Reference = No
Element Feature_PathDefinition (Type=axesgroupfeature)
  Type = PathDefinitions
    ModalDataBehaviour = UseAxesGroupSettings
    PathDefinition[1]:
      Name = Path1
      Type = CartesianPath
        CalculatedIn = PCS
      Limit = Internal
        Velocity = NotUsed
        Acceleration = NotUsed
        Deceleration = NotUsed
        Jerk = NotUsed
Element Feature_Tracking (Type=axesgroupfeature)
  Type = Tracking
    ModalDataBehaviour = UseAxesGroupSettings
    SynchronisationGeometry = Basic
      CartesianRadius = 20.0
```

### Rob1Ax.axis - ACP/mappMotion/Rob/Rob_1_4ax/Rob1Ax.axis
```
Element gR1_AxisQ1 (Type=axis)
  BaseTypeIsReadOnly = 0
  BaseType = RotaryBounded
    MeasurementUnitIsReadOnly = 0
    MeasurementUnit = 17476
    MeasurementResolutionIsReadOnly = 0
    MeasurementResolution = 0.01
    CountDirectionIsReadOnly = 0
    CountDirection = Inverse
  MovementLimitsIsReadOnly = 0
  MovementLimits = External
    LimitRef = LimitArm
  Alarms = None
Element gR1_AxisQ2 (Type=axis)
  BaseTypeIsReadOnly = 0
  BaseType = RotaryBounded
    MeasurementUnitIsReadOnly = 0
    MeasurementUnit = 17476
    MeasurementResolutionIsReadOnly = 0
    MeasurementResolution = 0.01
    CountDirectionIsReadOnly = 0
    CountDirection = Inverse
  MovementLimitsIsReadOnly = 0
  MovementLimits = External
    LimitRef = LimitArm
  Alarms = None
Element gR1_AxisQ3 (Type=axis)
  BaseTypeIsReadOnly = 0
  BaseType = RotaryBounded
    MeasurementUnitIsReadOnly = 0
    MeasurementUnit = 17476
    MeasurementResolutionIsReadOnly = 0
    MeasurementResolution = 0.01
    CountDirectionIsReadOnly = 0
    CountDirection = Inverse
  MovementLimitsIsReadOnly = 0
  MovementLimits = External
    LimitRef = LimitArm
  Alarms = None
Element gR1_AxisQC (Type=axis)
  BaseTypeIsReadOnly = 0
  BaseType = RotaryBounded
    MeasurementUnitIsReadOnly = 0
    MeasurementUnit = 17476
    MeasurementResolutionIsReadOnly = 0
    MeasurementResolution = 0.01
    CountDirectionIsReadOnly = 0
    CountDirection = Standard
  MovementLimitsIsReadOnly = 0
  MovementLimits = InternalForPathControlledAxis
    Position:
      LowerLimitMin = -1.79769313486231E308
      UpperLimitMax = 1.79769313486231E308
      LowerLimit = -170
      UpperLimit = 170
    VelocityIsReadOnly = 0
    Velocity:
      VelocityMax = 3.4E38
      Velocity = 1800
    AccelerationIsReadOnly = 0
    Acceleration:
      AccelerationMax = 3.4E38
      Acceleration = 9000
    DecelerationIsReadOnly = 0
    Deceleration:
      DecelerationMax = 3.4E38
      Deceleration = 9000
    JerkIsReadOnly = 0
    Jerk = Basic
      JerkMax = 3.4E38
      Jerk = 9000
    TorqueIsReadOnly = 0
  Alarms = None
Element gR1_AxisQA (Type=axis)
  BaseTypeIsReadOnly = 0
  BaseType = Rotary
    MeasurementUnitIsReadOnly = 0
    MeasurementUnit = 17476
    MeasurementResolutionIsReadOnly = 0
    MeasurementResolution = 0.01
    CountDirectionIsReadOnly = 0
    CountDirection = Standard
  MovementLimitsIsReadOnly = 0
  MovementLimits = External
    LimitRef = LimitTilt
  Alarms = None
```

### Rob1AxGr4.axesgroup - ACP/mappMotion/Rob/Rob_1_4ax/Rob1AxGr4.axesgroup
```
Element Rob1_4ax (Type=axesgroup)
  Type = PathGenAxesGroup
    ProcessingTaskClass = 1
    License = 1
    PhysicalAxes:
      JointAxes:
        JointAxis[1]:
          Name = Q1
          AxisRef = gR1_AxisQ1
        JointAxis[2]:
          Name = Q2
          AxisRef = gR1_AxisQ2
        JointAxis[3]:
          Name = Q3
          AxisRef = gR1_AxisQ3
        JointAxis[4]:
          Name = QC
          AxisRef = gR1_AxisQC
    MechanicalSystem:
      MechSysRef = MechSys_4ax
    BasicSettings:
      ModalDataBehaviour = ResetToDefault
      GeometryPlanning:
        TCPResolution:
          LengthResolution = 0.001
          AngleResolution = 0.001
        RoundingMode = Standard
        MaxCornerDeviation = 1
        MaxTangentialTransitionDeviation = 0.1
        MaxRadiusDeviation = 0.001
        WorkingPlane = XY
      TrajectoryPlanning = Basic
        LimitCheckResolution = UserDefinedTime
          Time = 0.005
        BufferTime = UserDefinedTime
          Time = 0.1
    AxesGroupFeatures:
      FeatureRef[1] = Feature_Programs
      FeatureRef[2] = Feature_Jogging
      FeatureRef[3] = Feature_PathDefinition
      FeatureRef[4] = Feature_Tracking
      FeatureRef[5] = Feature_FrameHierarchy
  Alarms = None
```

### Config_1.trackingpath - ACP/mappMotion/TrkPath/Config_1.trackingpath
```
Element gTrackingPath_Place_R1 (Type=trackingpath)
  Type = Linear
    MaxTrackingFrames = 50
    MotionSource = Axis
      AxisRef = gAxisConvB
  Alarms = MpAlarmX
Element gTrackingPath_Pick_R1 (Type=trackingpath)
  Type = Linear
    MaxTrackingFrames = 50
    MotionSource = Axis
      AxisRef = gAxisConvA
  Alarms = MpAlarmX
```

## Logical view

Binary libraries used (declarations not repeated): MTBasics 5.05.0, operator, runtime, astime, AsIecCon, DataObj, standard, AsArSdm, asstring, AsBrStr, MTTypes 1.03.4, brsystem, sys_lib, MTFilter 5.02.0, powerlnk, AsIODiag, AsBrMath, BRIT_Data 1.00.2, MpBase, McAcpAx 5.16.9, McAcpPar 5.16.9, McPathGen 5.16.9, McProgInt 5.16.9, McAcpTrak 5.16.9, McPureVAx 5.16.9, MpPick 5.16.9, McTrkPath 5.16.9, McPathSvc 5.16.9, MpAxis 5.16.9, McAxis 5.16.9, MpRobotics 5.16.9, McAxGroup 5.16.9, McBase 5.16.9, CoTrace 5.16.9, AsZip, FileIO

### Package Logical/Libraries - Global libraries

### Library Logical/Libraries/CamProf (ANSIC) - RONCHI - Cam profile calculations
Depends on: AsBrStr

#### CamProf.typ - Exported data types
```iecst
TYPE
	CamPolynomialData_typ : 	STRUCT
		a : REAL;
		b : REAL;
		c : REAL;
		d : REAL;
		e : REAL;
		f : REAL;
		g : REAL;
		x : REAL;
		Reserve : UDINT;
	END_STRUCT;
	CamProfile_typ : 	STRUCT
		MasterPeriod : DINT;
		SlavePeriod : DINT;
		PolynomialNumber : UDINT;
		PolynomialData : ARRAY[0..MAX_POLYNOMIALS_IDX]OF CamPolynomialData_typ;
	END_STRUCT;
END_TYPE

(**)

TYPE
	AddCamProf_par_typ : 	STRUCT
		master_start_add : REAL;
		master_add_distance : REAL;
		slave_add_distance : REAL;
		cam_end_position : REAL;
	END_STRUCT;
END_TYPE
```

#### CamProf.var - Exported constants
```iecst
VAR CONSTANT
	MAX_POLYNOMIALS_IDX : USINT := 127;
END_VAR
```

#### CamProf.fun - Exported functions and function blocks
```iecst
FUNCTION_BLOCK CamCalc (* *) (*$GROUP=User,$CAT=User,$GROUPICON=User.png,$CATICON=User.png*)
	VAR_INPUT
		Enable : BOOL;
		MasterSetSpeed : REAL;
		MasterActPosition : REAL;
		pCamPoly : REFERENCE TO CamProfile_typ;
		SL_Factor : REAL;
		MA_Factor : REAL;
	END_VAR
	VAR_OUTPUT
		SL_Acc : REAL;
		SL_Vel : REAL;
		SL_Pos : REAL;
		Valid : BOOL;
	END_VAR
	VAR
		xStart : REAL;
		x : ARRAY[0..6] OF REAL;
		poly : USINT;
		j : USINT;
		i : USINT;
	END_VAR
END_FUNCTION_BLOCK

{REDUND_ERROR} FUNCTION AddCamProf : BOOL (* *) (*$GROUP=User,$CAT=User,$GROUPICON=User.png,$CATICON=User.png*)
	VAR_INPUT
		adrCam : UDINT;
		adrParameter : UDINT;
	END_VAR
END_FUNCTION
```

- CamCalc.c (not readable text: treated as protected, skipped)

- AddCamProf.c (not readable text: treated as protected, skipped)

### Package Logical/Source - Including Source code and related objects

### Global.typ - Global data types
```iecst
(*********** Delta ***********)

TYPE
	DeltaCtrl_type : 	STRUCT
		Cmd : DeltaCtrlCmd_type;
		Status : DeltaCtrlStatus_type;
		Parameter : DeltaCtrlParameter_type;
	END_STRUCT;
	DeltaCtrlCmd_type : 	STRUCT
		PowerOn : BOOL;
		Home : BOOL;
		MoveProgram : BOOL;
		Stop : BOOL;
		ErrorReset : BOOL;
		Interrupt : BOOL;
		Continue : BOOL;
	END_STRUCT;
	DeltaCtrlStatus_type : 	STRUCT
		Active : BOOL;
		Error : BOOL;
		PowerOn : BOOL;
		IsHomed : BOOL;
		MoveActive : BOOL;
		MoveDone : BOOL;
		Stopped : BOOL;
		InMotion : BOOL;
		ProductPicked : BOOL;
		ProductPlaced : BOOL;
		MoveInterrupted : BOOL;
		ProductInRange : BOOL;
		InterruptStatus : McPrgInfoInterruptEnum;
		X : LREAL;
		Y : LREAL;
		Z : LREAL;
	END_STRUCT;
	DeltaCtrlParameter_type : 	STRUCT
		Override : REAL;
		DeltaPar : MpDelta4AxisParType;
	END_STRUCT;
END_TYPE

(*********** Conveyor ***********)

TYPE
	ConveyorCtrl_type : 	STRUCT
		Cmd : ConveyorCtrlCmd_type;
		Status : ConveyorCtrlStatus_type;
		Parameter : ConveyorCtrlParameter_type;
	END_STRUCT;
	ConveyorCtrlCmd_type : 	STRUCT
		PowerOn : BOOL;
		Home : BOOL;
		MoveAdditive : BOOL;
		MoveAbsolute : BOOL;
		MoveVelocity : BOOL;
		ErrorReset : BOOL;
		Stop : BOOL;
		Update : BOOL;
	END_STRUCT;
	ConveyorCtrlStatus_type : 	STRUCT
		Active : BOOL;
		Error : BOOL;
		PowerOn : BOOL;
		IsHomed : BOOL;
		MoveActive : BOOL;
		MoveDone : BOOL;
		Position : LREAL;
		Velocity : REAL;
		MovementLeft : LREAL;
		PosStartMovement : LREAL;
		UpdateDone : BOOL;
	END_STRUCT;
	ConveyorCtrlParameter_type : 	STRUCT
		ConveyorPar : MpAxisBasicParType;
	END_STRUCT;
END_TYPE
```

### Global.var - Global variables
```iecst
VAR
	gDeltaCtrl : DeltaCtrl_type;
	gConveyorBCtrl : ConveyorCtrl_type;
	gConveyorACtrl : ConveyorCtrl_type;
	gPlaceProduct : BOOL := FALSE;
	gPickProduct : BOOL := FALSE;
	JointAxisPos : ARRAY[0..3] OF LREAL := [4(0.0)];
	gRun : BOOL := FALSE;
	gPowerOn : BOOL := FALSE;
	PVIposition : ARRAY[0..6] OF LREAL;
END_VAR
```

### Package Logical/Source/Motion - Including tasks and objects related with motion (Robots, Conveyors)

### Package Logical/Source/Motion/RobotProgram - Robot program

### PickPlace.st
```iecst
	VAR CONSTANT

		WaitPos : McPointType := (Pos:=(X:=0,Y:=100,Z:=-800)); // in machine frame

		TransitionPos_DF : McPointType := (Pos:=(X:=-200,Y:=50,Z:=40)); // DF - Drop Frame
		TransitionPos_MF : McPointType := (Pos:=(X:=-70,Y:=120,Z:=-915)); // MF - Machine Frame
		TransitionPos_PF : McPointType := (Pos:=(X:=50,Y:=150,Z:=60)); 	// PF - Pick Frame

		PlaceOffsetPos : McPointType := (Pos:=(X:=0,Y:=0,Z:=30)); 		// in drop frame
		PlacePos : McPointType := (Pos:=(X:=0,Y:=0,Z:=10));

		PickOffsetPos : McPointType := (Pos:=(X:=0,Y:=0,Z:=30));		// in pick frame
		PickPos : McPointType := (Pos:=(X:=0,Y:=0,Z:=10));

	END_VAR

	VAR {AT 'ProductPla'}

		ChoosenPlaceFrame : McTrkFrmIdentType;
		PlacementSelected : BOOL;
		RunPickAndPlace : BOOL;

	END_VAR

	VAR {AT 'ProductDet'}

		ChoosenPickFrame : McTrkFrmIdentType;
		ProductSelected : BOOL;
		RunPickAndPlace : BOOL;

	END_VAR

	PROGRAM _MAIN

	Feedrate(50000);
	MoveL(WaitPos);
	TrackObject(ChoosenPickFrame, PickOffsetPos);
	MoveL(PickPos);
	WaitTime(1);
	ProductPicked := TRUE;
	MoveL(PickOffsetPos);
	MoveL(TransitionPos_PF);
//	WaitUntilFlush(ChoosenPlaceFrame <> 0); // causes a motion stop
	TrackObject(ChoosenPlaceFrame, PlaceOffsetPos);
	MoveL(PlacePos);
	ProductPlaced := TRUE;
	ProductPicked := FALSE;
	WaitTime(1);
	MoveL(PlaceOffsetPos);
	ProductPlaced := FALSE;
	TrackStop(MachineFrame, WaitPos);

	END_PROGRAM
```

### Program Logical/Source/Motion/DeltaCtrl (IEC)

#### Variables.var
```iecst
VAR
	DeltaRobot4Ax : MpDelta4Axis;
	JointQ2 : MpAxisBasic;
	JointQ3 : MpAxisBasic;
	JointQC : MpAxisBasic;
	JointQ1 : MpAxisBasic;
	JointPar : MpAxisBasicParType := (Homing:=(Mode:=mcHOMING_DEFAULT));
END_VAR
```

#### Main.st
```iecst
PROGRAM _INIT

	JointPar.Homing.Mode			:= mcHOMING_DIRECT;

	gDeltaCtrl.Parameter.Override	:= 100;
	gDeltaCtrl.Parameter.DeltaPar.ProgramName	:= 'PickPlace.st';

END_PROGRAM

PROGRAM _CYCLIC

	IF JointQ1.Active AND JointQ2.Active AND JointQ3.Active AND JointQC.Active THEN
		DeltaRobot4Ax.Enable		:= TRUE;
		DeltaRobot4Ax.MpLink 		:= ADR(Rob1_4ax);
		DeltaRobot4Ax.Parameters 	:= ADR(gDeltaCtrl.Parameter.DeltaPar);
		DeltaRobot4Ax.Override		:= gDeltaCtrl.Parameter.Override;
	END_IF;

	DeltaRobot4Ax.MoveProgram	:= gDeltaCtrl.Cmd.MoveProgram;
	DeltaRobot4Ax.Home			:= gDeltaCtrl.Cmd.Home;
	DeltaRobot4Ax.Power			:= gDeltaCtrl.Cmd.PowerOn;
	DeltaRobot4Ax.Stop			:= gDeltaCtrl.Cmd.Stop;
	DeltaRobot4Ax.ErrorReset	:= gDeltaCtrl.Cmd.ErrorReset;
	DeltaRobot4Ax.Interrupt		:= gDeltaCtrl.Cmd.Interrupt;
	DeltaRobot4Ax.Continue		:= gDeltaCtrl.Cmd.Continue;

	JointQ1.Enable 		:= TRUE;
	JointQ1.MpLink 		:= ADR(gR1_AxisQ1);
	JointQ1.Parameters 	:= ADR(JointPar);

	JointQ2.Enable 		:= TRUE;
	JointQ2.MpLink 		:= ADR(gR1_AxisQ2);
	JointQ2.Parameters 	:= ADR(JointPar);

	JointQ3.Enable 		:= TRUE;
	JointQ3.MpLink 		:= ADR(gR1_AxisQ3);
	JointQ3.Parameters 	:= ADR(JointPar);

	JointQC.Enable 		:= TRUE;
	JointQC.MpLink 		:= ADR(gR1_AxisQC);
	JointQC.Parameters 	:= ADR(JointPar);

	// Call of FUBs
	JointQ1();
	JointQ2();
	JointQ3();
	JointQC();
	DeltaRobot4Ax();

	IF EDGEPOS(gPickProduct) AND DeltaRobot4Ax.PowerOn AND DeltaRobot4Ax.IsHomed THEN
		gDeltaCtrl.Cmd.MoveProgram 	:= TRUE;
	END_IF;

	IF DeltaRobot4Ax.MoveDone AND gDeltaCtrl.Cmd.MoveProgram THEN
		gDeltaCtrl.Cmd.MoveProgram	:= FALSE;
	END_IF;

	// Update status parameter of ctrl structure
	gDeltaCtrl.Status.Active			:= DeltaRobot4Ax.Active;
	gDeltaCtrl.Status.Error				:= DeltaRobot4Ax.Error;
	gDeltaCtrl.Status.IsHomed			:= DeltaRobot4Ax.IsHomed;
	gDeltaCtrl.Status.MoveActive		:= DeltaRobot4Ax.MoveActive;
	gDeltaCtrl.Status.MoveDone			:= DeltaRobot4Ax.MoveDone;
	gDeltaCtrl.Status.PowerOn			:= DeltaRobot4Ax.PowerOn;
	gDeltaCtrl.Status.MoveInterrupted	:= DeltaRobot4Ax.MoveInterrupted;
	gDeltaCtrl.Status.Stopped			:= DeltaRobot4Ax.Stopped;
	gDeltaCtrl.Status.InMotion			:= DeltaRobot4Ax.InMotion;
	gDeltaCtrl.Status.InterruptStatus	:= DeltaRobot4Ax.Info.Program.InterruptStatus;
	gDeltaCtrl.Status.X                 := DeltaRobot4Ax.X;
	gDeltaCtrl.Status.Y                 := DeltaRobot4Ax.Y;
	gDeltaCtrl.Status.Z                 := DeltaRobot4Ax.Z;

	JointAxisPos[0] := ( DeltaRobot4Ax.Info.JointAxisPosition[0] );
	JointAxisPos[1] := ( DeltaRobot4Ax.Info.JointAxisPosition[1] );
	JointAxisPos[2] := ( DeltaRobot4Ax.Info.JointAxisPosition[2] );
	JointAxisPos[3] := ( DeltaRobot4Ax.Info.JointAxisPosition[3] );

END_PROGRAM

PROGRAM _EXIT

	DeltaRobot4Ax.Enable	:= FALSE;
	DeltaRobot4Ax();
	JointQ1.Enable			:= FALSE;
	JointQ1();
	JointQ2.Enable			:= FALSE;
	JointQ2();
	JointQ3.Enable			:= FALSE;
	JointQ3();
	JointQC.Enable			:= FALSE;
	JointQC();

END_PROGRAM
```

### Program Logical/Source/Motion/ConveyorA (IEC)

#### Variables.var
```iecst
VAR
	Conveyor : MpAxisBasic;
END_VAR
```

#### Main.st
```iecst
PROGRAM _INIT

END_PROGRAM

PROGRAM _CYCLIC

	Conveyor.Enable 	:= TRUE;
	Conveyor.MpLink 	:= ADR(gAxisConvA);
	Conveyor.Parameters := ADR(gConveyorACtrl.Parameter.ConveyorPar);

	Conveyor.Power			:= gConveyorACtrl.Cmd.PowerOn;
	Conveyor.Home			:= gConveyorACtrl.Cmd.Home;
	Conveyor.ErrorReset		:= gConveyorACtrl.Cmd.ErrorReset;
	Conveyor.MoveAdditive	:= gConveyorACtrl.Cmd.MoveAdditive;
	Conveyor.MoveAbsolute	:= gConveyorACtrl.Cmd.MoveAbsolute;
	Conveyor.MoveVelocity	:= gConveyorACtrl.Cmd.MoveVelocity;
	Conveyor.Update			:= gConveyorACtrl.Cmd.Update;
	Conveyor.Stop			:= gConveyorACtrl.Cmd.Stop;

	IF EDGEPOS(Conveyor.MoveAdditive) THEN
		gConveyorACtrl.Status.PosStartMovement	:= Conveyor.Position;
		gConveyorACtrl.Cmd.MoveAdditive := FALSE;
	END_IF;

	Conveyor();

	gConveyorACtrl.Status.MovementLeft	:= (gConveyorACtrl.Status.PosStartMovement + gConveyorACtrl.Parameter.ConveyorPar.Distance) - Conveyor.Position;
	gConveyorACtrl.Status.Active		:= Conveyor.Active;
	gConveyorACtrl.Status.Error			:= Conveyor.Error;
	gConveyorACtrl.Status.IsHomed		:= Conveyor.IsHomed;
	gConveyorACtrl.Status.UpdateDone	:= Conveyor.UpdateDone;
	gConveyorACtrl.Status.MoveActive	:= Conveyor.MoveActive;
	gConveyorACtrl.Status.MoveDone		:= Conveyor.MoveDone;
	gConveyorACtrl.Status.PowerOn		:= Conveyor.PowerOn;
	gConveyorACtrl.Status.Position		:= Conveyor.Position;
	gConveyorACtrl.Status.Velocity		:= Conveyor.Velocity;

END_PROGRAM

PROGRAM _EXIT

	Conveyor.Enable 	:= FALSE;
	Conveyor();

END_PROGRAM
```

### Program Logical/Source/Motion/ConveyorB (IEC)

#### Main.st
```iecst
PROGRAM _INIT

END_PROGRAM

PROGRAM _CYCLIC

	Conveyor.Enable 	:= TRUE;
	Conveyor.MpLink 	:= ADR(gAxisConvB);
	Conveyor.Parameters := ADR(gConveyorBCtrl.Parameter.ConveyorPar);

	Conveyor.Power			:= gConveyorBCtrl.Cmd.PowerOn;
	Conveyor.Home			:= gConveyorBCtrl.Cmd.Home;
	Conveyor.ErrorReset		:= gConveyorBCtrl.Cmd.ErrorReset;
	Conveyor.MoveAdditive	:= gConveyorBCtrl.Cmd.MoveAdditive;
	Conveyor.MoveAbsolute	:= gConveyorBCtrl.Cmd.MoveAbsolute;
	Conveyor.MoveVelocity	:= gConveyorBCtrl.Cmd.MoveVelocity;
	Conveyor.Update			:= gConveyorBCtrl.Cmd.Update;
	Conveyor.Stop			:= gConveyorBCtrl.Cmd.Stop;

	IF EDGEPOS(Conveyor.MoveAdditive) THEN
		gConveyorBCtrl.Status.PosStartMovement	:= Conveyor.Position;
		gConveyorBCtrl.Cmd.MoveAdditive := FALSE;
	END_IF;

	Conveyor();

	gConveyorBCtrl.Status.MovementLeft	:= (gConveyorBCtrl.Status.PosStartMovement + gConveyorBCtrl.Parameter.ConveyorPar.Distance) - Conveyor.Position;
	gConveyorBCtrl.Status.Active		:= Conveyor.Active;
	gConveyorBCtrl.Status.Error			:= Conveyor.Error;
	gConveyorBCtrl.Status.IsHomed		:= Conveyor.IsHomed;
	gConveyorBCtrl.Status.UpdateDone	:= Conveyor.UpdateDone;
	gConveyorBCtrl.Status.MoveActive	:= Conveyor.MoveActive;
	gConveyorBCtrl.Status.MoveDone		:= Conveyor.MoveDone;
	gConveyorBCtrl.Status.PowerOn		:= Conveyor.PowerOn;
	gConveyorBCtrl.Status.Position		:= Conveyor.Position;
	gConveyorBCtrl.Status.Velocity		:= Conveyor.Velocity;

END_PROGRAM

PROGRAM _EXIT

	Conveyor.Enable 	:= FALSE;
	Conveyor();

END_PROGRAM
```

### Program Logical/Source/Motion/ProductDetect (IEC)

#### Variables.var
```iecst
VAR
	ProductSelected : BOOL := FALSE;
	MC_BR_TrackingFrameCreateManual : MC_BR_TrackingFrameCreate;
	MC_BR_TrackingPathGetFrames_Pick : MC_BR_TrackingPathGetFrames := (0);
	TrkFrmInfo : McTrkFrmInfoType := (0);
	TRF_Id_Manual : McTrkFrmIdentType := (0);
	ManualCreateFrame : BOOL := FALSE;
	ChoosenPickFrame : McTrkFrmIdentType := (0);
	ManualFrameX : LREAL := 0.0;
	ManualFrameY : LREAL := 0;
	DeleteFrame : BOOL := FALSE;
	MC_BR_TrackingFrameDelete_0 : MC_BR_TrackingFrameDelete := (0);
	RunPickAndPlace : BOOL;
	ProductPicked : BOOL;
	ProductPlaced : BOOL;
END_VAR
```

#### Main.st
```iecst
PROGRAM _INIT

	ProductSelected;
	ChoosenPickFrame;
	RunPickAndPlace	:= TRUE;
	gConveyorACtrl.Parameter.ConveyorPar.Acceleration	:= 200;
	gConveyorACtrl.Parameter.ConveyorPar.Deceleration	:= 200;
	gConveyorACtrl.Parameter.ConveyorPar.Distance		:= -400;
	gConveyorACtrl.Parameter.ConveyorPar.Velocity		:= 50;
	ManualFrameX	:= 0;
	ManualFrameY	:= 0;

END_PROGRAM

PROGRAM _CYCLIC

	IF gPowerOn THEN
		gDeltaCtrl.Cmd.Home	:= TRUE;
		gDeltaCtrl.Cmd.PowerOn	:= TRUE;
		gConveyorACtrl.Cmd.Home	:= TRUE;
		gConveyorACtrl.Cmd.PowerOn	:= TRUE;
	END_IF;

	IF EDGEPOS(gRun) THEN
		ManualCreateFrame := TRUE;
		gConveyorACtrl.Cmd.MoveVelocity := TRUE;
	END_IF

	IF ManualCreateFrame AND TRF_Id_Manual = 0 THEN
		gDeltaCtrl.Status.ProductPlaced := FALSE;
		MC_BR_TrackingFrameCreateManual.Execute	:= TRUE;
		MC_BR_TrackingFrameCreateManual.Parameters.Translation.X			:= ManualFrameX;
		MC_BR_TrackingFrameCreateManual.Parameters.Translation.Y			:= ManualFrameY;
		MC_BR_TrackingFrameCreateManual.Parameters.Translation.Z			:= -985;
		MC_BR_TrackingFrameCreateManual.Parameters.LatchedPath.Position	:= gConveyorACtrl.Status.Position;
		MC_BR_TrackingFrameCreateManual.TrackingPath	:= ADR(gTrackingPath_Pick_R1);
		IF MC_BR_TrackingFrameCreateManual.Done THEN
			MC_BR_TrackingFrameCreateManual.Execute	:= FALSE;
			ManualCreateFrame	:= FALSE;
			TRF_Id_Manual	:= MC_BR_TrackingFrameCreateManual.TrackingFrameID;
		END_IF;
	END_IF;

	MC_BR_TrackingFrameCreateManual();

	ProductPlaced := gDeltaCtrl.Status.ProductPlaced;

	IF TRF_Id_Manual <> 0 THEN
		MC_BR_TrackingPathGetFrames_Pick.Execute		:= TRUE;
		MC_BR_TrackingPathGetFrames_Pick.TrackingPath		:= ADR(gTrackingPath_Pick_R1);
		MC_BR_TrackingPathGetFrames_Pick.Parameters.DataAddress	:= ADR(TrkFrmInfo);
		MC_BR_TrackingPathGetFrames_Pick.Parameters.NumberOfFrames	:= 1;
		MC_BR_TrackingPathGetFrames_Pick.Parameters.GetMode	:= mcTRKPATH_GET_MOD_ALL_FRAMES;
		MC_BR_TrackingPathGetFrames_Pick();
		IF MC_BR_TrackingPathGetFrames_Pick.Done THEN
			IF (TrkFrmInfo.Distance > 400 AND TrkFrmInfo.Distance < 800 AND NOT ProductPlaced)  THEN
				ProductSelected	:= TRUE;
				ChoosenPickFrame	:= TrkFrmInfo.TrackingFrameID;
			ELSIF (*TrkFrmInfo.Distance > 800 OR *)ProductPlaced THEN
				ProductSelected		:= FALSE;
				ChoosenPickFrame	:= 0;
				DeleteFrame			:= TRUE;
			END_IF;
			MC_BR_TrackingPathGetFrames_Pick.Execute		:= FALSE;
			MC_BR_TrackingPathGetFrames_Pick();
		END_IF;
	END_IF;

	IF DeleteFrame THEN
		MC_BR_TrackingFrameDelete_0.Execute			:= TRUE;
		MC_BR_TrackingFrameDelete_0.Mode			:= mcTRKFRM_DELETE_MOD_ALL;
		MC_BR_TrackingFrameDelete_0.TrackingPath	:= ADR(gTrackingPath_Pick_R1);
		MC_BR_TrackingFrameDelete_0();
		IF MC_BR_TrackingFrameDelete_0.Done THEN
			MC_BR_TrackingFrameDelete_0.Execute	:= FALSE;
			DeleteFrame		:= FALSE;
			ManualCreateFrame := TRUE;
			TRF_Id_Manual	:= 0;
			MC_BR_TrackingFrameDelete_0();
		END_IF;
	END_IF;

	gPickProduct	:= ProductSelected;

	ProductPicked;
	ProductPlaced;

	PVIposition[0] := JointAxisPos[0];
	PVIposition[1] := JointAxisPos[1];
	PVIposition[2] := JointAxisPos[2];
	PVIposition[3] := JointAxisPos[3];
	PVIposition[4] := TrkFrmInfo.CurrentPosition.X -605;
	PVIposition[5] := TrkFrmInfo.CurrentPosition.Y;
	PVIposition[6] := -20;

END_PROGRAM

PROGRAM _EXIT
	(* Insert code here *)

END_PROGRAM
```

### Program Logical/Source/Motion/ProductPlacement (IEC)

#### Variables.var
```iecst
VAR
	PlacementSelected : BOOL := FALSE;
	MC_BR_TrackingFrameCreateManual : MC_BR_TrackingFrameCreate;
	MC_BR_TrackingPathGetFrames_Plce : MC_BR_TrackingPathGetFrames := (0);
	TrkFrmInfo : McTrkFrmInfoType := (0);
	TRF_Id_Manual : McTrkFrmIdentType := (0);
	ManualCreateFrame : BOOL := FALSE;
	ChoosenPlaceFrame : McTrkFrmIdentType := (0);
	ManualFrameX : LREAL := 0.0;
	ManualFrameY : LREAL := 0;
	DeleteFrame : BOOL := FALSE;
	MC_BR_TrackingFrameDelete_0 : MC_BR_TrackingFrameDelete := (0);
	RunPickAndPlace : BOOL;
	ProductPicked : BOOL;
	ProductPlaced : BOOL;
END_VAR
```

#### Main.st
```iecst
PROGRAM _INIT

	PlacementSelected;
	ChoosenPlaceFrame;
	RunPickAndPlace	:= TRUE;
	gConveyorBCtrl.Parameter.ConveyorPar.Acceleration	:= 200;
	gConveyorBCtrl.Parameter.ConveyorPar.Deceleration	:= 200;
	gConveyorBCtrl.Parameter.ConveyorPar.Distance		:= -400;
	gConveyorBCtrl.Parameter.ConveyorPar.Velocity		:= 5;
	ManualFrameX	:= 0;
	ManualFrameY	:= 0;

END_PROGRAM

PROGRAM _CYCLIC

	IF gPowerOn THEN
		gDeltaCtrl.Cmd.Home	:= TRUE;
		gDeltaCtrl.Cmd.PowerOn	:= TRUE;
		gConveyorBCtrl.Cmd.Home	:= TRUE;
		gConveyorBCtrl.Cmd.PowerOn	:= TRUE;
	END_IF;

	IF EDGEPOS(gRun) THEN
		ManualCreateFrame := TRUE;
	END_IF

	IF ManualCreateFrame AND TRF_Id_Manual = 0 THEN
		gDeltaCtrl.Status.ProductPlaced := FALSE;
		MC_BR_TrackingFrameCreateManual.Execute	:= TRUE;
		MC_BR_TrackingFrameCreateManual.Parameters.Translation.X			:= ManualFrameX;
		MC_BR_TrackingFrameCreateManual.Parameters.Translation.Y			:= ManualFrameY;
		MC_BR_TrackingFrameCreateManual.Parameters.Translation.Z			:= -985;
		MC_BR_TrackingFrameCreateManual.Parameters.LatchedPath.Position	:= gConveyorBCtrl.Status.Position;
		MC_BR_TrackingFrameCreateManual.TrackingPath	:= ADR(gTrackingPath_Place_R1);
		IF MC_BR_TrackingFrameCreateManual.Done THEN
			MC_BR_TrackingFrameCreateManual.Execute	:= FALSE;
			ManualCreateFrame	:= FALSE;
			TRF_Id_Manual	:= MC_BR_TrackingFrameCreateManual.TrackingFrameID;
		END_IF;
	END_IF;

	MC_BR_TrackingFrameCreateManual();

	ProductPlaced := gDeltaCtrl.Status.ProductPlaced;

	IF TRF_Id_Manual <> 0 THEN
		MC_BR_TrackingPathGetFrames_Plce.Execute		:= TRUE;
		MC_BR_TrackingPathGetFrames_Plce.TrackingPath		:= ADR(gTrackingPath_Place_R1);
		MC_BR_TrackingPathGetFrames_Plce.Parameters.DataAddress	:= ADR(TrkFrmInfo);
		MC_BR_TrackingPathGetFrames_Plce.Parameters.NumberOfFrames	:= 1;
		MC_BR_TrackingPathGetFrames_Plce.Parameters.GetMode	:= mcTRKPATH_GET_MOD_ALL_FRAMES;

		IF MC_BR_TrackingPathGetFrames_Plce.Done THEN
			IF (TrkFrmInfo.Distance >= 0 AND TrkFrmInfo.Distance < 800)  THEN
				PlacementSelected	:= TRUE;
				ChoosenPlaceFrame	:= TrkFrmInfo.TrackingFrameID;
			ELSIF (*TrkFrmInfo.Distance > 800 OR *)ProductPlaced THEN
				PlacementSelected		:= FALSE;
				ChoosenPlaceFrame	:= 0;
				DeleteFrame			:= TRUE;
			END_IF;
			MC_BR_TrackingPathGetFrames_Plce.Execute		:= FALSE;
	//		MC_BR_TrackingPathGetFrames_Plce();
		END_IF;
	END_IF;

	IF DeleteFrame THEN
		MC_BR_TrackingFrameDelete_0.Execute			:= TRUE;
		MC_BR_TrackingFrameDelete_0.Mode			:= mcTRKFRM_DELETE_MOD_ALL;
		MC_BR_TrackingFrameDelete_0.TrackingPath	:= ADR(gTrackingPath_Place_R1);
//		MC_BR_TrackingFrameDelete_0();
		IF MC_BR_TrackingFrameDelete_0.Done THEN
			MC_BR_TrackingFrameDelete_0.Execute	:= FALSE;
			DeleteFrame		:= FALSE;
	//		ManualCreateFrame := TRUE;
			TRF_Id_Manual	:= 0;

		END_IF;
	END_IF;

	gPlaceProduct	:= PlacementSelected;

	MC_BR_TrackingPathGetFrames_Plce();
	MC_BR_TrackingFrameDelete_0();
	ProductPicked;
	ProductPlaced;

//	PVIposition[0] := JointAxisPos[0];
//	PVIposition[1] := JointAxisPos[1];
//	PVIposition[2] := JointAxisPos[2];
//	PVIposition[3] := JointAxisPos[3];
//	PVIposition[4] := TrkFrmInfo.CurrentPosition.X -605;
//	PVIposition[5] := TrkFrmInfo.CurrentPosition.Y;
//	PVIposition[6] := -20;

END_PROGRAM

PROGRAM _EXIT
	(* Insert code here *)

END_PROGRAM
```

### Package Logical/Source/Simulation - Including Tasks related with the robotic visualization (simulation of the process)

- TrackingSampleDocumentation.docx (binary file, 901828 bytes)
Listed in the project but not available here: Logical/Variables.var, Logical/Types.typ
